(*
	Link component with additional interface:
	Control BYTE: From TwinCAT >>> To Unity	(Default)
	Status BYTE: FROM Unity >>> TO TwinCAT	(Default)
	ControlData LWORD: From TwinCAT >>> To Unity		
	StatusData LWORD: FROM Unity >>> TO TwinCAT		
*)
FUNCTION_BLOCK FB_LinkDataLWord EXTENDS FB_LinkDevice
VAR	
	{attribute 'simulation_interface'}
	ControlData		AT %Q* : LWORD;
	{attribute 'simulation_interface'}
	StatusData		AT %I* : LWORD;
END_VAR

SUPER^();

METHOD INTERNAL GetLinkControlData : LWORD
GetLinkControlData := ControlData;
END_METHOD

METHOD INTERNAL SetLinkStatusData : BOOL
VAR_INPUT
	nStatusData : LWORD;
END_VAR
StatusData := nStatusData;
END_METHOD

END_FUNCTION_BLOCK

(* stored: Version 1.1.0.1, ProductVersion 3.1.4024.12
   POU FB_LinkDataLWord: Id {1972ec6c-e9f1-0295-1c53-5bd7bae6e40c}, SpecialFunc None
   Method GetLinkControlData: Id {68aa099c-6f15-0510-3e8b-1c6ed923ba6b}
   Method SetLinkStatusData: Id {e9556268-4f18-099e-3cf7-1fdb5bb0087e} *)
